// TIA Portal project "Aufgabe_1_002_mCopilot" (V20)
// *** This TIA Portal project underwent AI modifications via the Siemens Engineering Copilot. ***

(* hardware
DEVICE "S7-1500/ET200MP-Station_1"  S7-1500 station
   slot 0: "Profilschiene_0"  Rack  6ES7 590-1***0-0AA0
   slot 1: "PLC_1"  CPU 1512C-1 PN  6ES7 512-1CK01-0AB0  V2.9
      slot 3: "CPU-Display_1"  6ES7591-1AA00-0AA0
      slot 32768: "PROFINET-Schnittstelle_1"  X1
         slot 32769: "Port_1"  X1 P1
         slot 32770: "Port_2"  X1 P2
      slot 34817: "Virtual CP interface port_1"  Virtual CP interface port  Virtual CP interface port
*)

// ===== PLC "PLC_1"  CPU 1512C-1 PN =====

VAR_GLOBAL   // PLC tag table "Standard-Variablentabelle"
   "x_Start_Prozess" AT %M0.0 : Bool;
   "x_Abgeschlossen" AT %M0.1 : Bool;
END_VAR

VAR_GLOBAL   // PLC tag table "Stanzmaschine"
   "x_Lichtschranke_Ein_Auslagerung" AT %I0.0 : Bool;   // 0 = Werkstueck vorhanden (Oeffner)
   "x_Lichtschranke_Stanzposition" AT %I0.1 : Bool;   // 0 = Werkstueck vorhanden (Oeffner)
   "x_Endlage_Stanze_oben" AT %I0.2 : Bool;   // 1 = Stanze oben (Schliesser)
   "x_Endlage_Stanze_unten" AT %I0.3 : Bool;   // 1 = Stanze oben (Schliesser)
   "x_Motor_Transportband_Vorwaerts" AT %Q0.0 : Bool;   // 1 = Motor laeuft
   "x_Motor_Transportband_Rueckwaerts" AT %Q0.1 : Bool;   // 1 = Motor laeuft
   "x_Motor_Stanze_nach_oben" AT %Q0.2 : Bool;   // 1 = Stanze faehrt aufwaerts
   "x_Motor_Stanze_nach_unten" AT %Q0.3 : Bool;   // 1 = Stanze faehrt abwaerts
END_VAR

TYPE "ST_Werkzeug"
   STRUCT
      i_Werkzeug_ID : Int;
      i_Haltezeit_ms : Int;
      x_Aktiv : Bool;
   END_STRUCT;
END_TYPE

DATA_BLOCK "FB_Stanzprozess_erweitert_DB"   // DB1
{ S7_Optimized_Access := 'TRUE' }
VERSION : 0.1
// stored: InstanceOfName FB_Stanzprozess_erweitert
"FB_Stanzprozess_erweitert"
BEGIN
END_DATA_BLOCK

DATA_BLOCK "Test_DB"   // DB2
{ S7_Optimized_Access := 'TRUE' }
VERSION : 0.1
   VAR
      x_Start_Prozess : Bool;
      x_Fertig : Bool;
      stWerkzeug_Werkzeug_1_Daten : "ST_Werkzeug";
      stWerkzeug_Werkzeug_2_Daten : "ST_Werkzeug";
      stWerkzeug_Werkzeug_3_Daten : "ST_Werkzeug";
      iArray_Anzahl_Stanzvorgaenge : Array[0..4] of Int;
      i_Status : Int;
   END_VAR
BEGIN
   stWerkzeug_Werkzeug_1_Daten.i_Werkzeug_ID := 1;
   stWerkzeug_Werkzeug_1_Daten.i_Haltezeit_ms := 500;
   stWerkzeug_Werkzeug_2_Daten.i_Werkzeug_ID := 2;
   stWerkzeug_Werkzeug_2_Daten.i_Haltezeit_ms := 200;
   stWerkzeug_Werkzeug_3_Daten.i_Werkzeug_ID := 3;
   stWerkzeug_Werkzeug_3_Daten.i_Haltezeit_ms := 900;
END_DATA_BLOCK

FUNCTION_BLOCK "FB_Stanzprozess_erweitert"   // FB12, SCL
{ S7_Optimized_Access := 'TRUE' }
VERSION : 0.1
   VAR_INPUT
      x_Ausfuehren : Bool;
      x_Stanze_oben : Bool;
      x_Stanze_unten : Bool;
      stWerkzeug_Werkzeugdaten : "ST_Werkzeug";
   END_VAR
   VAR_OUTPUT
      x_Fertig : Bool;
      x_Stanze_hoch : Bool;
      x_Stanze_runter : Bool;
      i_Status : Int;
   END_VAR
   VAR_IN_OUT
      iArray_Stanzzaehler : Array[0..4] of Int;
   END_VAR
   VAR
      x_Prozess_aktiv : Bool;
      x_Abwaerts_fertig : Bool;
      x_Haltezeit_aktiv : Bool;
      x_Aufwaerts_fertig : Bool;
      x_Ausfuehren_alt : Bool;
      x_Flanke : Bool;
      time_TON_Haltezeit : TON_TIME;
      time_Aktuelle_Haltezeit : Time;
      i_Werkzeug_Index : Int;
   END_VAR
BEGIN

   REGION INFO HEADER
       //===============================================================================
       //-------------------------------------------------------------------------------
       // Title:            FB_Stanzprozess_erweitert
       // Comment/Function: Dieser Funktionsbaustein steuert die vertikale Bewegung der Stanz und implementiert
       //                   zusaetzliche Funktionen fuer die Statusueberwachung, flexible Werkzeugparameter
       //                   und Produktionserfassung. Der Stanzprozess kann mit bis zu 5 verschiedenen
       //                   Werkzeugen gesteuert werden. Jedes dieser Werkzeuge wird durch eine eindeutige
       //                   Werkzeug_ID im bereich von 0 bis 4 identifiziert. Welches Werkzeug genutzt werden
       //                   soll, wird dem Baustein ueber die Eingangsvariable stWerkzeug_Werkzeugdaten uebermittelt.
       // Library/Family:   N.A
       // Author:           ---
       // Tested with:      S7-1500 CPU 1512C-1 PN DC/DC/DC FW 2.9
       // Engineering:      TIA Portal V20
       // Requirements:     --- 
       //-------------------------------------------------------------------------------
       // Change log table:
       // Version  | Date       | Expert in charge        | Changes applied
       //----------|------------|-------------------------|-----------------------------
       // 01.00.00 | 10.12.2025 |          N.N            | First released version
       //===============================================================================
   END_REGION INFO HEADER

   REGION PROCESS
       #x_Flanke := #x_Ausfuehren AND NOT #x_Ausfuehren_alt;
       #x_Ausfuehren_alt := #x_Ausfuehren;

       #time_Aktuelle_Haltezeit := INT_TO_TIME(#stWerkzeug_Werkzeugdaten.i_Haltezeit_ms);
       #i_Werkzeug_Index := #stWerkzeug_Werkzeugdaten.i_Werkzeug_ID;

       IF #x_Flanke AND NOT #x_Prozess_aktiv THEN
           #x_Prozess_aktiv := TRUE;
           #x_Fertig := FALSE;
           #x_Abwaerts_fertig := FALSE;
           #x_Haltezeit_aktiv := FALSE;
           #x_Aufwaerts_fertig := FALSE;
           #i_Status := 1;
       END_IF;

       IF #x_Prozess_aktiv THEN

           IF NOT #x_Abwaerts_fertig THEN
               #x_Stanze_runter := TRUE;
               #x_Stanze_hoch := FALSE;
               #i_Status := 1;

               IF #x_Stanze_unten THEN
                   #x_Stanze_runter := FALSE;
                   #x_Abwaerts_fertig := TRUE;
                   #x_Haltezeit_aktiv := TRUE;
                   #i_Status := 2;
               END_IF
           END_IF;

           #time_TON_Haltezeit_(IN := #x_Haltezeit_aktiv,          
                               PT := #time_Aktuelle_Haltezeit);

           IF #time_TON_Haltezeit.Q AND #x_Haltezeit_aktiv THEN
               #x_Haltezeit_aktiv := FALSE;
               #i_Status := 3;
           END_IF;

           IF #x_Abwaerts_fertig AND NOT #x_Haltezeit_aktiv AND NOT #x_Aufwaerts_fertig THEN
               #x_Stanze_hoch := TRUE;
               #x_Stanze_runter := FALSE;

               IF #x_Stanze_oben THEN
                   #x_Stanze_hoch := FALSE;
                   #x_Aufwaerts_fertig := TRUE;
                   #i_Status := 4;
               END_IF;
           END_IF;

           IF #x_Aufwaerts_fertig THEN
               #x_Fertig := TRUE;
               #i_Status := 4;
           END_IF;

           IF #i_Werkzeug_Index >= 0 AND #i_Werkzeug_Index <= 4 THEN
               #iArray_Stanzzaehler[#i_Werkzeug_Index] := #iArray_Stanzzaehler[#i_Werkzeug_Index] + 1;
           END_IF;

           IF #x_Fertig THEN
               #x_Prozess_aktiv := FALSE;
           END_IF;

       ELSE
           #x_Stanze_hoch := FALSE;
           #x_Stanze_runter := FALSE;
           IF NOT #x_Fertig THEN
               #i_Status := 0;
           END_IF;
       END_IF;

   END_REGION PROCESS
END_FUNCTION_BLOCK

FUNCTION "FC_Check" : Void   // FC1, SCL
{ S7_Optimized_Access := 'TRUE' }
VERSION : 0.1
BEGIN
   //Funktionsinhalt nur zur Ueberpruefung der korrekten Verknuepfung des Projekts,
   //mit dem Engineering Copilot
   //
   //Rechenaufgabe
   //Berechne das Produkt von 8 und 4
END_FUNCTION

ORGANIZATION_BLOCK "Main"   // OB1, FBD, ProgramCycle
TITLE = "Main Program Sweep (Cycle)"
{ S7_Optimized_Access := 'TRUE' }
VERSION : 0.1
   VAR_INPUT
      Initial_Call : Bool;   // Initial call of this OB
      Remanence : Bool;   // =True, if remanent data are available
   END_VAR
BEGIN

REGION Network 1: FB_Stanzprozess_erweitert
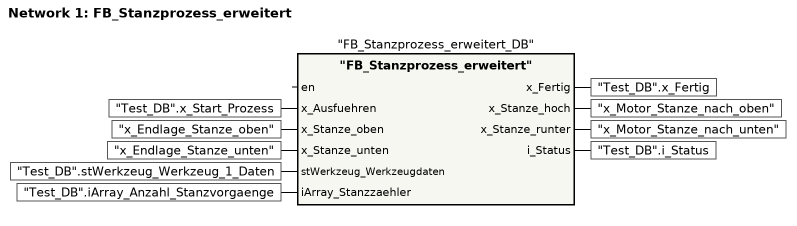
   "FB_Stanzprozess_erweitert_DB"(x_Ausfuehren := "Test_DB".x_Start_Prozess,   // "FB_Stanzprozess_erweitert"
                           x_Stanze_oben := "x_Endlage_Stanze_oben",
                           x_Stanze_unten := "x_Endlage_Stanze_unten",
                           stWerkzeug_Werkzeugdaten := "Test_DB".stWerkzeug_Werkzeug_1_Daten,
                           iArray_Stanzzaehler := "Test_DB".iArray_Anzahl_Stanzvorgaenge,
                           x_Fertig => "Test_DB".x_Fertig,
                           x_Stanze_hoch => "x_Motor_Stanze_nach_oben",
                           x_Stanze_runter => "x_Motor_Stanze_nach_unten",
                           i_Status => "Test_DB".i_Status);
END_REGION
END_ORGANIZATION_BLOCK